// TIA Portal V20 export
TYPE "typeSequenceControlNodeHomeCheck_sideTapeLoading"
// stored: Namespace Unit1.Em4
   STRUCT
      TapeLoadReq { ExternalWritable := 'False'} : Bool;
      TapeLoaded { ExternalWritable := 'False'} : Bool;
   END_STRUCT;
END_TYPE
